// TIA Portal V18 export
FUNCTION "PLC8_910A4_8DI_8DO_IO_Update" : Void   // FC11070, LAD
{ S7_Optimized_Access := 'TRUE' }
VERSION : 0.1
// stored: AutoNumber false, IsIECCheckEnabled false, SetENOAutomatically false, UDAEnableTagReadback false
BEGIN

REGION Network 1: DIa0
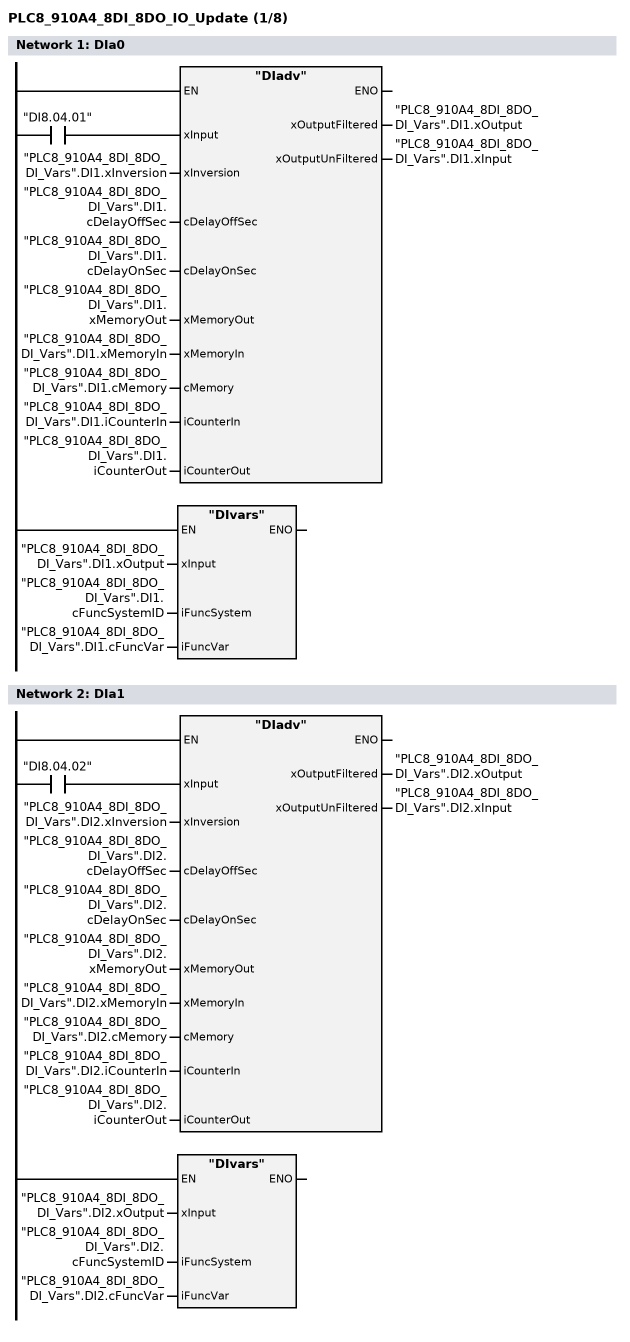
   RUNG wire#powerrail
      "DIadv"(xInput := wire#w1, xInversion := "PLC8_910A4_8DI_8DO_DI_Vars".DI1.xInversion, cDelayOffSec := "PLC8_910A4_8DI_8DO_DI_Vars".DI1.cDelayOffSec, cDelayOnSec := "PLC8_910A4_8DI_8DO_DI_Vars".DI1.cDelayOnSec, xMemoryOut := "PLC8_910A4_8DI_8DO_DI_Vars".DI1.xMemoryOut, xMemoryIn := "PLC8_910A4_8DI_8DO_DI_Vars".DI1.xMemoryIn, cMemory := "PLC8_910A4_8DI_8DO_DI_Vars".DI1.cMemory, iCounterIn := "PLC8_910A4_8DI_8DO_DI_Vars".DI1.iCounterIn, iCounterOut := "PLC8_910A4_8DI_8DO_DI_Vars".DI1.iCounterOut, xOutputFiltered => "PLC8_910A4_8DI_8DO_DI_Vars".DI1.xOutput, xOutputUnFiltered => "PLC8_910A4_8DI_8DO_DI_Vars".DI1.xInput)
   END_RUNG
   RUNG wire#powerrail
      Contact( "DI8.04.01" )
   END_RUNG wire#w1
   RUNG wire#powerrail
      "DIvars"(xInput := "PLC8_910A4_8DI_8DO_DI_Vars".DI1.xOutput, iFuncSystem := "PLC8_910A4_8DI_8DO_DI_Vars".DI1.cFuncSystemID, iFuncVar := "PLC8_910A4_8DI_8DO_DI_Vars".DI1.cFuncVar)
   END_RUNG
   // the same network as SCL:
   "DIadv"(xInput := "DI8.04.01",
           xInversion := "PLC8_910A4_8DI_8DO_DI_Vars".DI1.xInversion,
           cDelayOffSec := "PLC8_910A4_8DI_8DO_DI_Vars".DI1.cDelayOffSec,
           cDelayOnSec := "PLC8_910A4_8DI_8DO_DI_Vars".DI1.cDelayOnSec,
           xMemoryOut := "PLC8_910A4_8DI_8DO_DI_Vars".DI1.xMemoryOut,
           xMemoryIn := "PLC8_910A4_8DI_8DO_DI_Vars".DI1.xMemoryIn,
           cMemory := "PLC8_910A4_8DI_8DO_DI_Vars".DI1.cMemory,
           iCounterIn := "PLC8_910A4_8DI_8DO_DI_Vars".DI1.iCounterIn,
           iCounterOut := "PLC8_910A4_8DI_8DO_DI_Vars".DI1.iCounterOut,
           xOutputFiltered => "PLC8_910A4_8DI_8DO_DI_Vars".DI1.xOutput,
           xOutputUnFiltered => "PLC8_910A4_8DI_8DO_DI_Vars".DI1.xInput);
   "DIvars"(xInput := "PLC8_910A4_8DI_8DO_DI_Vars".DI1.xOutput,
            iFuncSystem := "PLC8_910A4_8DI_8DO_DI_Vars".DI1.cFuncSystemID,
            iFuncVar := "PLC8_910A4_8DI_8DO_DI_Vars".DI1.cFuncVar);
END_REGION

REGION Network 2: DIa1
   RUNG wire#powerrail
      "DIadv"(xInput := wire#w1, xInversion := "PLC8_910A4_8DI_8DO_DI_Vars".DI2.xInversion, cDelayOffSec := "PLC8_910A4_8DI_8DO_DI_Vars".DI2.cDelayOffSec, cDelayOnSec := "PLC8_910A4_8DI_8DO_DI_Vars".DI2.cDelayOnSec, xMemoryOut := "PLC8_910A4_8DI_8DO_DI_Vars".DI2.xMemoryOut, xMemoryIn := "PLC8_910A4_8DI_8DO_DI_Vars".DI2.xMemoryIn, cMemory := "PLC8_910A4_8DI_8DO_DI_Vars".DI2.cMemory, iCounterIn := "PLC8_910A4_8DI_8DO_DI_Vars".DI2.iCounterIn, iCounterOut := "PLC8_910A4_8DI_8DO_DI_Vars".DI2.iCounterOut, xOutputFiltered => "PLC8_910A4_8DI_8DO_DI_Vars".DI2.xOutput, xOutputUnFiltered => "PLC8_910A4_8DI_8DO_DI_Vars".DI2.xInput)
   END_RUNG
   RUNG wire#powerrail
      Contact( "DI8.04.02" )
   END_RUNG wire#w1
   RUNG wire#powerrail
      "DIvars"(xInput := "PLC8_910A4_8DI_8DO_DI_Vars".DI2.xOutput, iFuncSystem := "PLC8_910A4_8DI_8DO_DI_Vars".DI2.cFuncSystemID, iFuncVar := "PLC8_910A4_8DI_8DO_DI_Vars".DI2.cFuncVar)
   END_RUNG
   // the same network as SCL:
   "DIadv"(xInput := "DI8.04.02",
           xInversion := "PLC8_910A4_8DI_8DO_DI_Vars".DI2.xInversion,
           cDelayOffSec := "PLC8_910A4_8DI_8DO_DI_Vars".DI2.cDelayOffSec,
           cDelayOnSec := "PLC8_910A4_8DI_8DO_DI_Vars".DI2.cDelayOnSec,
           xMemoryOut := "PLC8_910A4_8DI_8DO_DI_Vars".DI2.xMemoryOut,
           xMemoryIn := "PLC8_910A4_8DI_8DO_DI_Vars".DI2.xMemoryIn,
           cMemory := "PLC8_910A4_8DI_8DO_DI_Vars".DI2.cMemory,
           iCounterIn := "PLC8_910A4_8DI_8DO_DI_Vars".DI2.iCounterIn,
           iCounterOut := "PLC8_910A4_8DI_8DO_DI_Vars".DI2.iCounterOut,
           xOutputFiltered => "PLC8_910A4_8DI_8DO_DI_Vars".DI2.xOutput,
           xOutputUnFiltered => "PLC8_910A4_8DI_8DO_DI_Vars".DI2.xInput);
   "DIvars"(xInput := "PLC8_910A4_8DI_8DO_DI_Vars".DI2.xOutput,
            iFuncSystem := "PLC8_910A4_8DI_8DO_DI_Vars".DI2.cFuncSystemID,
            iFuncVar := "PLC8_910A4_8DI_8DO_DI_Vars".DI2.cFuncVar);
END_REGION

REGION Network 3: DIa2
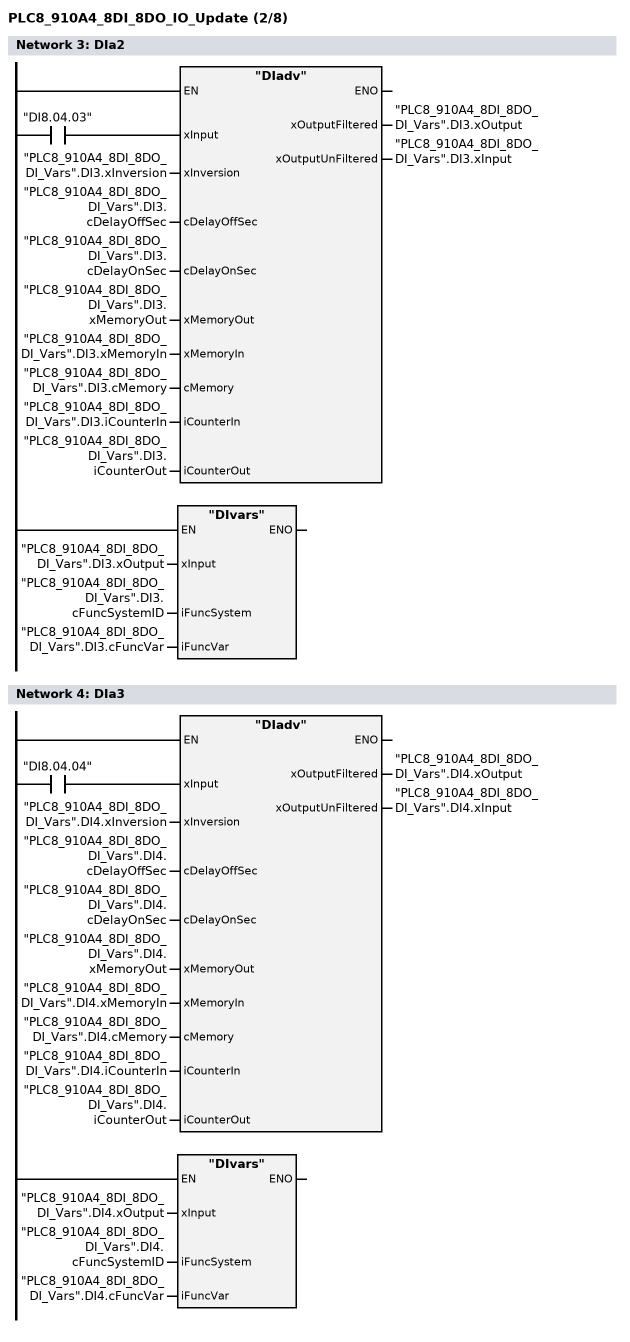
   RUNG wire#powerrail
      "DIadv"(xInput := wire#w1, xInversion := "PLC8_910A4_8DI_8DO_DI_Vars".DI3.xInversion, cDelayOffSec := "PLC8_910A4_8DI_8DO_DI_Vars".DI3.cDelayOffSec, cDelayOnSec := "PLC8_910A4_8DI_8DO_DI_Vars".DI3.cDelayOnSec, xMemoryOut := "PLC8_910A4_8DI_8DO_DI_Vars".DI3.xMemoryOut, xMemoryIn := "PLC8_910A4_8DI_8DO_DI_Vars".DI3.xMemoryIn, cMemory := "PLC8_910A4_8DI_8DO_DI_Vars".DI3.cMemory, iCounterIn := "PLC8_910A4_8DI_8DO_DI_Vars".DI3.iCounterIn, iCounterOut := "PLC8_910A4_8DI_8DO_DI_Vars".DI3.iCounterOut, xOutputFiltered => "PLC8_910A4_8DI_8DO_DI_Vars".DI3.xOutput, xOutputUnFiltered => "PLC8_910A4_8DI_8DO_DI_Vars".DI3.xInput)
   END_RUNG
   RUNG wire#powerrail
      Contact( "DI8.04.03" )
   END_RUNG wire#w1
   RUNG wire#powerrail
      "DIvars"(xInput := "PLC8_910A4_8DI_8DO_DI_Vars".DI3.xOutput, iFuncSystem := "PLC8_910A4_8DI_8DO_DI_Vars".DI3.cFuncSystemID, iFuncVar := "PLC8_910A4_8DI_8DO_DI_Vars".DI3.cFuncVar)
   END_RUNG
   // the same network as SCL:
   "DIadv"(xInput := "DI8.04.03",
           xInversion := "PLC8_910A4_8DI_8DO_DI_Vars".DI3.xInversion,
           cDelayOffSec := "PLC8_910A4_8DI_8DO_DI_Vars".DI3.cDelayOffSec,
           cDelayOnSec := "PLC8_910A4_8DI_8DO_DI_Vars".DI3.cDelayOnSec,
           xMemoryOut := "PLC8_910A4_8DI_8DO_DI_Vars".DI3.xMemoryOut,
           xMemoryIn := "PLC8_910A4_8DI_8DO_DI_Vars".DI3.xMemoryIn,
           cMemory := "PLC8_910A4_8DI_8DO_DI_Vars".DI3.cMemory,
           iCounterIn := "PLC8_910A4_8DI_8DO_DI_Vars".DI3.iCounterIn,
           iCounterOut := "PLC8_910A4_8DI_8DO_DI_Vars".DI3.iCounterOut,
           xOutputFiltered => "PLC8_910A4_8DI_8DO_DI_Vars".DI3.xOutput,
           xOutputUnFiltered => "PLC8_910A4_8DI_8DO_DI_Vars".DI3.xInput);
   "DIvars"(xInput := "PLC8_910A4_8DI_8DO_DI_Vars".DI3.xOutput,
            iFuncSystem := "PLC8_910A4_8DI_8DO_DI_Vars".DI3.cFuncSystemID,
            iFuncVar := "PLC8_910A4_8DI_8DO_DI_Vars".DI3.cFuncVar);
END_REGION

REGION Network 4: DIa3
   RUNG wire#powerrail
      "DIadv"(xInput := wire#w1, xInversion := "PLC8_910A4_8DI_8DO_DI_Vars".DI4.xInversion, cDelayOffSec := "PLC8_910A4_8DI_8DO_DI_Vars".DI4.cDelayOffSec, cDelayOnSec := "PLC8_910A4_8DI_8DO_DI_Vars".DI4.cDelayOnSec, xMemoryOut := "PLC8_910A4_8DI_8DO_DI_Vars".DI4.xMemoryOut, xMemoryIn := "PLC8_910A4_8DI_8DO_DI_Vars".DI4.xMemoryIn, cMemory := "PLC8_910A4_8DI_8DO_DI_Vars".DI4.cMemory, iCounterIn := "PLC8_910A4_8DI_8DO_DI_Vars".DI4.iCounterIn, iCounterOut := "PLC8_910A4_8DI_8DO_DI_Vars".DI4.iCounterOut, xOutputFiltered => "PLC8_910A4_8DI_8DO_DI_Vars".DI4.xOutput, xOutputUnFiltered => "PLC8_910A4_8DI_8DO_DI_Vars".DI4.xInput)
   END_RUNG
   RUNG wire#powerrail
      Contact( "DI8.04.04" )
   END_RUNG wire#w1
   RUNG wire#powerrail
      "DIvars"(xInput := "PLC8_910A4_8DI_8DO_DI_Vars".DI4.xOutput, iFuncSystem := "PLC8_910A4_8DI_8DO_DI_Vars".DI4.cFuncSystemID, iFuncVar := "PLC8_910A4_8DI_8DO_DI_Vars".DI4.cFuncVar)
   END_RUNG
   // the same network as SCL:
   "DIadv"(xInput := "DI8.04.04",
           xInversion := "PLC8_910A4_8DI_8DO_DI_Vars".DI4.xInversion,
           cDelayOffSec := "PLC8_910A4_8DI_8DO_DI_Vars".DI4.cDelayOffSec,
           cDelayOnSec := "PLC8_910A4_8DI_8DO_DI_Vars".DI4.cDelayOnSec,
           xMemoryOut := "PLC8_910A4_8DI_8DO_DI_Vars".DI4.xMemoryOut,
           xMemoryIn := "PLC8_910A4_8DI_8DO_DI_Vars".DI4.xMemoryIn,
           cMemory := "PLC8_910A4_8DI_8DO_DI_Vars".DI4.cMemory,
           iCounterIn := "PLC8_910A4_8DI_8DO_DI_Vars".DI4.iCounterIn,
           iCounterOut := "PLC8_910A4_8DI_8DO_DI_Vars".DI4.iCounterOut,
           xOutputFiltered => "PLC8_910A4_8DI_8DO_DI_Vars".DI4.xOutput,
           xOutputUnFiltered => "PLC8_910A4_8DI_8DO_DI_Vars".DI4.xInput);
   "DIvars"(xInput := "PLC8_910A4_8DI_8DO_DI_Vars".DI4.xOutput,
            iFuncSystem := "PLC8_910A4_8DI_8DO_DI_Vars".DI4.cFuncSystemID,
            iFuncVar := "PLC8_910A4_8DI_8DO_DI_Vars".DI4.cFuncVar);
END_REGION

REGION Network 5: DIa4
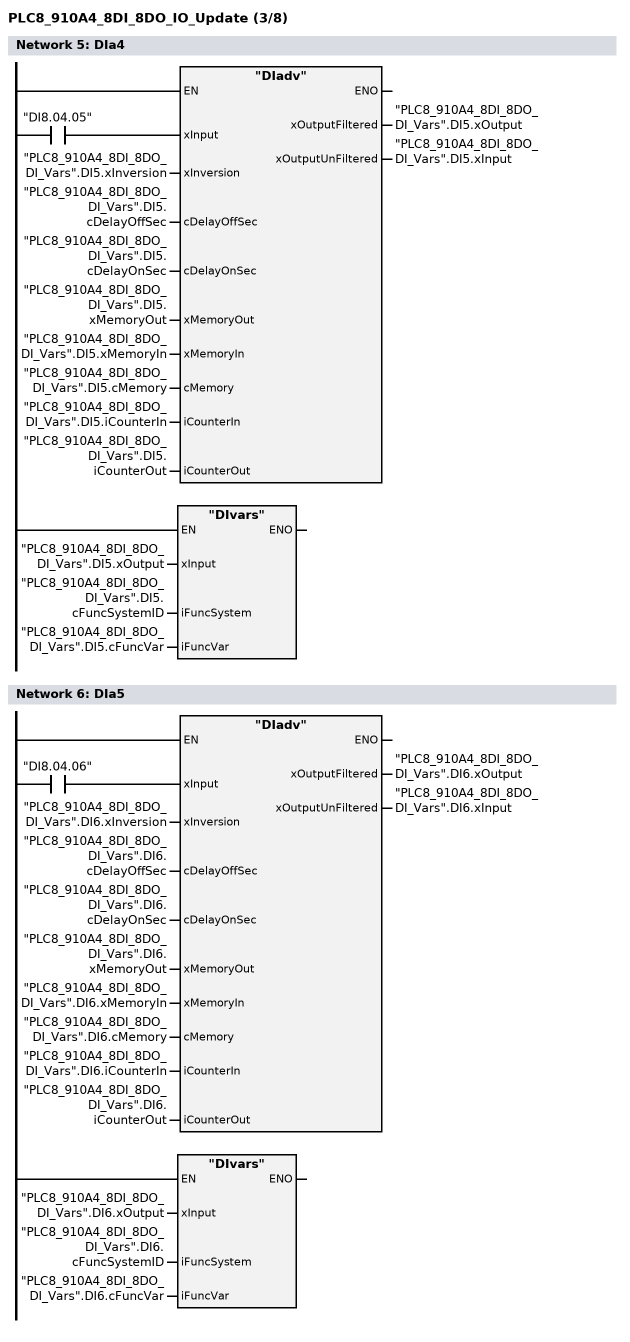
   RUNG wire#powerrail
      "DIadv"(xInput := wire#w1, xInversion := "PLC8_910A4_8DI_8DO_DI_Vars".DI5.xInversion, cDelayOffSec := "PLC8_910A4_8DI_8DO_DI_Vars".DI5.cDelayOffSec, cDelayOnSec := "PLC8_910A4_8DI_8DO_DI_Vars".DI5.cDelayOnSec, xMemoryOut := "PLC8_910A4_8DI_8DO_DI_Vars".DI5.xMemoryOut, xMemoryIn := "PLC8_910A4_8DI_8DO_DI_Vars".DI5.xMemoryIn, cMemory := "PLC8_910A4_8DI_8DO_DI_Vars".DI5.cMemory, iCounterIn := "PLC8_910A4_8DI_8DO_DI_Vars".DI5.iCounterIn, iCounterOut := "PLC8_910A4_8DI_8DO_DI_Vars".DI5.iCounterOut, xOutputFiltered => "PLC8_910A4_8DI_8DO_DI_Vars".DI5.xOutput, xOutputUnFiltered => "PLC8_910A4_8DI_8DO_DI_Vars".DI5.xInput)
   END_RUNG
   RUNG wire#powerrail
      Contact( "DI8.04.05" )
   END_RUNG wire#w1
   RUNG wire#powerrail
      "DIvars"(xInput := "PLC8_910A4_8DI_8DO_DI_Vars".DI5.xOutput, iFuncSystem := "PLC8_910A4_8DI_8DO_DI_Vars".DI5.cFuncSystemID, iFuncVar := "PLC8_910A4_8DI_8DO_DI_Vars".DI5.cFuncVar)
   END_RUNG
   // the same network as SCL:
   "DIadv"(xInput := "DI8.04.05",
           xInversion := "PLC8_910A4_8DI_8DO_DI_Vars".DI5.xInversion,
           cDelayOffSec := "PLC8_910A4_8DI_8DO_DI_Vars".DI5.cDelayOffSec,
           cDelayOnSec := "PLC8_910A4_8DI_8DO_DI_Vars".DI5.cDelayOnSec,
           xMemoryOut := "PLC8_910A4_8DI_8DO_DI_Vars".DI5.xMemoryOut,
           xMemoryIn := "PLC8_910A4_8DI_8DO_DI_Vars".DI5.xMemoryIn,
           cMemory := "PLC8_910A4_8DI_8DO_DI_Vars".DI5.cMemory,
           iCounterIn := "PLC8_910A4_8DI_8DO_DI_Vars".DI5.iCounterIn,
           iCounterOut := "PLC8_910A4_8DI_8DO_DI_Vars".DI5.iCounterOut,
           xOutputFiltered => "PLC8_910A4_8DI_8DO_DI_Vars".DI5.xOutput,
           xOutputUnFiltered => "PLC8_910A4_8DI_8DO_DI_Vars".DI5.xInput);
   "DIvars"(xInput := "PLC8_910A4_8DI_8DO_DI_Vars".DI5.xOutput,
            iFuncSystem := "PLC8_910A4_8DI_8DO_DI_Vars".DI5.cFuncSystemID,
            iFuncVar := "PLC8_910A4_8DI_8DO_DI_Vars".DI5.cFuncVar);
END_REGION

REGION Network 6: DIa5
   RUNG wire#powerrail
      "DIadv"(xInput := wire#w1, xInversion := "PLC8_910A4_8DI_8DO_DI_Vars".DI6.xInversion, cDelayOffSec := "PLC8_910A4_8DI_8DO_DI_Vars".DI6.cDelayOffSec, cDelayOnSec := "PLC8_910A4_8DI_8DO_DI_Vars".DI6.cDelayOnSec, xMemoryOut := "PLC8_910A4_8DI_8DO_DI_Vars".DI6.xMemoryOut, xMemoryIn := "PLC8_910A4_8DI_8DO_DI_Vars".DI6.xMemoryIn, cMemory := "PLC8_910A4_8DI_8DO_DI_Vars".DI6.cMemory, iCounterIn := "PLC8_910A4_8DI_8DO_DI_Vars".DI6.iCounterIn, iCounterOut := "PLC8_910A4_8DI_8DO_DI_Vars".DI6.iCounterOut, xOutputFiltered => "PLC8_910A4_8DI_8DO_DI_Vars".DI6.xOutput, xOutputUnFiltered => "PLC8_910A4_8DI_8DO_DI_Vars".DI6.xInput)
   END_RUNG
   RUNG wire#powerrail
      Contact( "DI8.04.06" )
   END_RUNG wire#w1
   RUNG wire#powerrail
      "DIvars"(xInput := "PLC8_910A4_8DI_8DO_DI_Vars".DI6.xOutput, iFuncSystem := "PLC8_910A4_8DI_8DO_DI_Vars".DI6.cFuncSystemID, iFuncVar := "PLC8_910A4_8DI_8DO_DI_Vars".DI6.cFuncVar)
   END_RUNG
   // the same network as SCL:
   "DIadv"(xInput := "DI8.04.06",
           xInversion := "PLC8_910A4_8DI_8DO_DI_Vars".DI6.xInversion,
           cDelayOffSec := "PLC8_910A4_8DI_8DO_DI_Vars".DI6.cDelayOffSec,
           cDelayOnSec := "PLC8_910A4_8DI_8DO_DI_Vars".DI6.cDelayOnSec,
           xMemoryOut := "PLC8_910A4_8DI_8DO_DI_Vars".DI6.xMemoryOut,
           xMemoryIn := "PLC8_910A4_8DI_8DO_DI_Vars".DI6.xMemoryIn,
           cMemory := "PLC8_910A4_8DI_8DO_DI_Vars".DI6.cMemory,
           iCounterIn := "PLC8_910A4_8DI_8DO_DI_Vars".DI6.iCounterIn,
           iCounterOut := "PLC8_910A4_8DI_8DO_DI_Vars".DI6.iCounterOut,
           xOutputFiltered => "PLC8_910A4_8DI_8DO_DI_Vars".DI6.xOutput,
           xOutputUnFiltered => "PLC8_910A4_8DI_8DO_DI_Vars".DI6.xInput);
   "DIvars"(xInput := "PLC8_910A4_8DI_8DO_DI_Vars".DI6.xOutput,
            iFuncSystem := "PLC8_910A4_8DI_8DO_DI_Vars".DI6.cFuncSystemID,
            iFuncVar := "PLC8_910A4_8DI_8DO_DI_Vars".DI6.cFuncVar);
END_REGION

REGION Network 7: DIa6
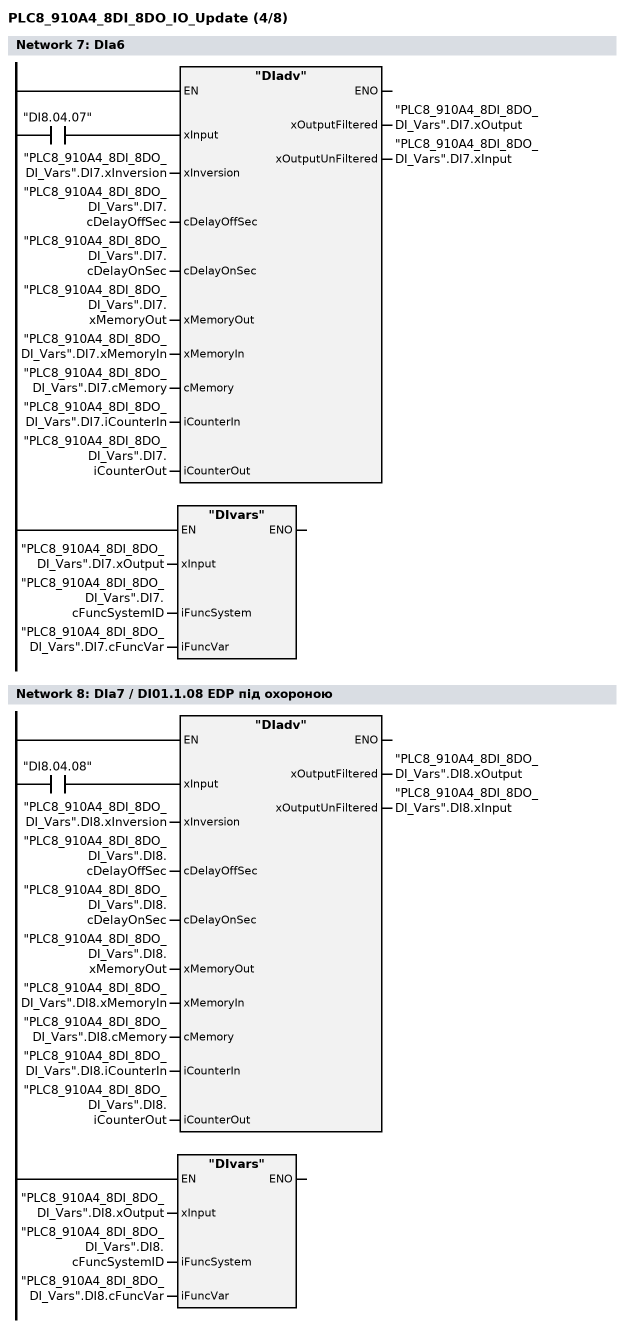
   RUNG wire#powerrail
      "DIadv"(xInput := wire#w1, xInversion := "PLC8_910A4_8DI_8DO_DI_Vars".DI7.xInversion, cDelayOffSec := "PLC8_910A4_8DI_8DO_DI_Vars".DI7.cDelayOffSec, cDelayOnSec := "PLC8_910A4_8DI_8DO_DI_Vars".DI7.cDelayOnSec, xMemoryOut := "PLC8_910A4_8DI_8DO_DI_Vars".DI7.xMemoryOut, xMemoryIn := "PLC8_910A4_8DI_8DO_DI_Vars".DI7.xMemoryIn, cMemory := "PLC8_910A4_8DI_8DO_DI_Vars".DI7.cMemory, iCounterIn := "PLC8_910A4_8DI_8DO_DI_Vars".DI7.iCounterIn, iCounterOut := "PLC8_910A4_8DI_8DO_DI_Vars".DI7.iCounterOut, xOutputFiltered => "PLC8_910A4_8DI_8DO_DI_Vars".DI7.xOutput, xOutputUnFiltered => "PLC8_910A4_8DI_8DO_DI_Vars".DI7.xInput)
   END_RUNG
   RUNG wire#powerrail
      Contact( "DI8.04.07" )
   END_RUNG wire#w1
   RUNG wire#powerrail
      "DIvars"(xInput := "PLC8_910A4_8DI_8DO_DI_Vars".DI7.xOutput, iFuncSystem := "PLC8_910A4_8DI_8DO_DI_Vars".DI7.cFuncSystemID, iFuncVar := "PLC8_910A4_8DI_8DO_DI_Vars".DI7.cFuncVar)
   END_RUNG
   // the same network as SCL:
   "DIadv"(xInput := "DI8.04.07",
           xInversion := "PLC8_910A4_8DI_8DO_DI_Vars".DI7.xInversion,
           cDelayOffSec := "PLC8_910A4_8DI_8DO_DI_Vars".DI7.cDelayOffSec,
           cDelayOnSec := "PLC8_910A4_8DI_8DO_DI_Vars".DI7.cDelayOnSec,
           xMemoryOut := "PLC8_910A4_8DI_8DO_DI_Vars".DI7.xMemoryOut,
           xMemoryIn := "PLC8_910A4_8DI_8DO_DI_Vars".DI7.xMemoryIn,
           cMemory := "PLC8_910A4_8DI_8DO_DI_Vars".DI7.cMemory,
           iCounterIn := "PLC8_910A4_8DI_8DO_DI_Vars".DI7.iCounterIn,
           iCounterOut := "PLC8_910A4_8DI_8DO_DI_Vars".DI7.iCounterOut,
           xOutputFiltered => "PLC8_910A4_8DI_8DO_DI_Vars".DI7.xOutput,
           xOutputUnFiltered => "PLC8_910A4_8DI_8DO_DI_Vars".DI7.xInput);
   "DIvars"(xInput := "PLC8_910A4_8DI_8DO_DI_Vars".DI7.xOutput,
            iFuncSystem := "PLC8_910A4_8DI_8DO_DI_Vars".DI7.cFuncSystemID,
            iFuncVar := "PLC8_910A4_8DI_8DO_DI_Vars".DI7.cFuncVar);
END_REGION

REGION Network 8: DIa7 / DI01.1.08 EDP під охороною
   RUNG wire#powerrail
      "DIadv"(xInput := wire#w1, xInversion := "PLC8_910A4_8DI_8DO_DI_Vars".DI8.xInversion, cDelayOffSec := "PLC8_910A4_8DI_8DO_DI_Vars".DI8.cDelayOffSec, cDelayOnSec := "PLC8_910A4_8DI_8DO_DI_Vars".DI8.cDelayOnSec, xMemoryOut := "PLC8_910A4_8DI_8DO_DI_Vars".DI8.xMemoryOut, xMemoryIn := "PLC8_910A4_8DI_8DO_DI_Vars".DI8.xMemoryIn, cMemory := "PLC8_910A4_8DI_8DO_DI_Vars".DI8.cMemory, iCounterIn := "PLC8_910A4_8DI_8DO_DI_Vars".DI8.iCounterIn, iCounterOut := "PLC8_910A4_8DI_8DO_DI_Vars".DI8.iCounterOut, xOutputFiltered => "PLC8_910A4_8DI_8DO_DI_Vars".DI8.xOutput, xOutputUnFiltered => "PLC8_910A4_8DI_8DO_DI_Vars".DI8.xInput)
   END_RUNG
   RUNG wire#powerrail
      Contact( "DI8.04.08" )
   END_RUNG wire#w1
   RUNG wire#powerrail
      "DIvars"(xInput := "PLC8_910A4_8DI_8DO_DI_Vars".DI8.xOutput, iFuncSystem := "PLC8_910A4_8DI_8DO_DI_Vars".DI8.cFuncSystemID, iFuncVar := "PLC8_910A4_8DI_8DO_DI_Vars".DI8.cFuncVar)
   END_RUNG
   // the same network as SCL:
   "DIadv"(xInput := "DI8.04.08",
           xInversion := "PLC8_910A4_8DI_8DO_DI_Vars".DI8.xInversion,
           cDelayOffSec := "PLC8_910A4_8DI_8DO_DI_Vars".DI8.cDelayOffSec,
           cDelayOnSec := "PLC8_910A4_8DI_8DO_DI_Vars".DI8.cDelayOnSec,
           xMemoryOut := "PLC8_910A4_8DI_8DO_DI_Vars".DI8.xMemoryOut,
           xMemoryIn := "PLC8_910A4_8DI_8DO_DI_Vars".DI8.xMemoryIn,
           cMemory := "PLC8_910A4_8DI_8DO_DI_Vars".DI8.cMemory,
           iCounterIn := "PLC8_910A4_8DI_8DO_DI_Vars".DI8.iCounterIn,
           iCounterOut := "PLC8_910A4_8DI_8DO_DI_Vars".DI8.iCounterOut,
           xOutputFiltered => "PLC8_910A4_8DI_8DO_DI_Vars".DI8.xOutput,
           xOutputUnFiltered => "PLC8_910A4_8DI_8DO_DI_Vars".DI8.xInput);
   "DIvars"(xInput := "PLC8_910A4_8DI_8DO_DI_Vars".DI8.xOutput,
            iFuncSystem := "PLC8_910A4_8DI_8DO_DI_Vars".DI8.cFuncSystemID,
            iFuncVar := "PLC8_910A4_8DI_8DO_DI_Vars".DI8.cFuncVar);
END_REGION

REGION Network 9: DQa0
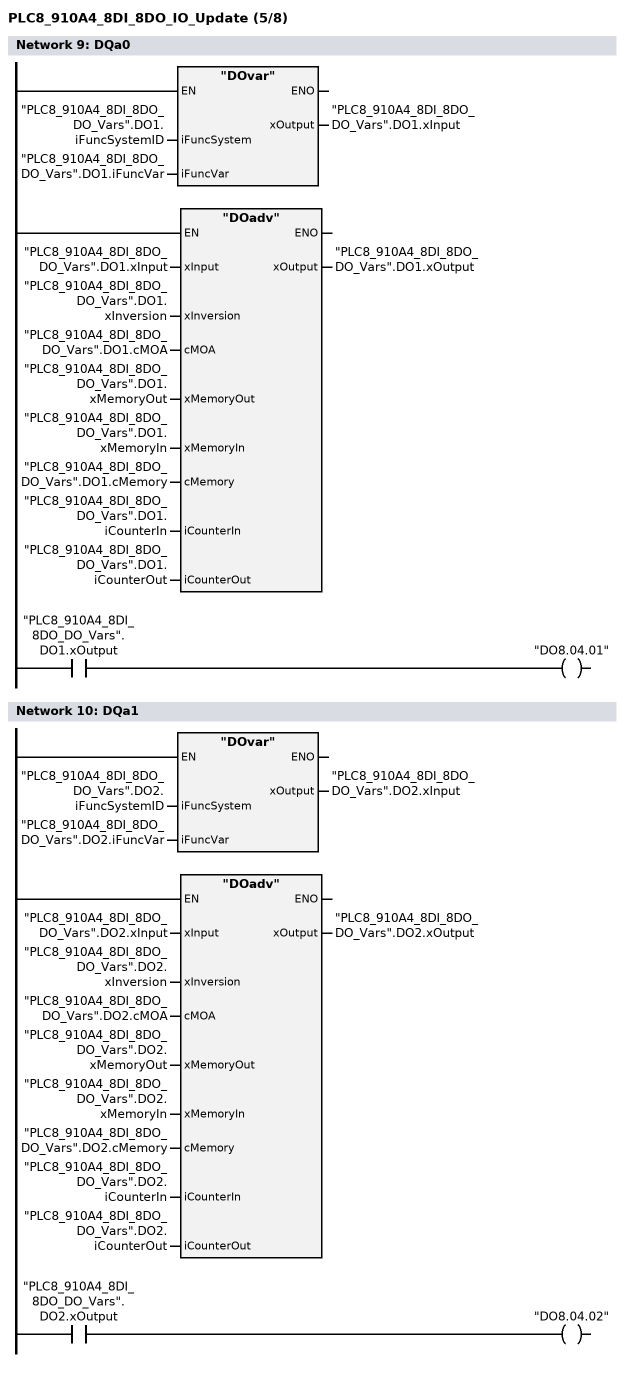
   RUNG wire#powerrail
      "DOvar"(iFuncSystem := "PLC8_910A4_8DI_8DO_DO_Vars".DO1.iFuncSystemID, iFuncVar := "PLC8_910A4_8DI_8DO_DO_Vars".DO1.iFuncVar, xOutput => "PLC8_910A4_8DI_8DO_DO_Vars".DO1.xInput)
   END_RUNG
   RUNG wire#powerrail
      "DOadv"(xInput := "PLC8_910A4_8DI_8DO_DO_Vars".DO1.xInput, xInversion := "PLC8_910A4_8DI_8DO_DO_Vars".DO1.xInversion, cMOA := "PLC8_910A4_8DI_8DO_DO_Vars".DO1.cMOA, xMemoryOut := "PLC8_910A4_8DI_8DO_DO_Vars".DO1.xMemoryOut, xMemoryIn := "PLC8_910A4_8DI_8DO_DO_Vars".DO1.xMemoryIn, cMemory := "PLC8_910A4_8DI_8DO_DO_Vars".DO1.cMemory, iCounterIn := "PLC8_910A4_8DI_8DO_DO_Vars".DO1.iCounterIn, iCounterOut := "PLC8_910A4_8DI_8DO_DO_Vars".DO1.iCounterOut, xOutput => "PLC8_910A4_8DI_8DO_DO_Vars".DO1.xOutput)
   END_RUNG
   RUNG wire#powerrail
      Contact( "PLC8_910A4_8DI_8DO_DO_Vars".DO1.xOutput )
      Coil( "DO8.04.01" )
   END_RUNG
   // the same network as SCL:
   "DOvar"(iFuncSystem := "PLC8_910A4_8DI_8DO_DO_Vars".DO1.iFuncSystemID,
           iFuncVar := "PLC8_910A4_8DI_8DO_DO_Vars".DO1.iFuncVar,
           xOutput => "PLC8_910A4_8DI_8DO_DO_Vars".DO1.xInput);
   "DOadv"(xInput := "PLC8_910A4_8DI_8DO_DO_Vars".DO1.xInput,
           xInversion := "PLC8_910A4_8DI_8DO_DO_Vars".DO1.xInversion,
           cMOA := "PLC8_910A4_8DI_8DO_DO_Vars".DO1.cMOA,
           xMemoryOut := "PLC8_910A4_8DI_8DO_DO_Vars".DO1.xMemoryOut,
           xMemoryIn := "PLC8_910A4_8DI_8DO_DO_Vars".DO1.xMemoryIn,
           cMemory := "PLC8_910A4_8DI_8DO_DO_Vars".DO1.cMemory,
           iCounterIn := "PLC8_910A4_8DI_8DO_DO_Vars".DO1.iCounterIn,
           iCounterOut := "PLC8_910A4_8DI_8DO_DO_Vars".DO1.iCounterOut,
           xOutput => "PLC8_910A4_8DI_8DO_DO_Vars".DO1.xOutput);
   "DO8.04.01" := "PLC8_910A4_8DI_8DO_DO_Vars".DO1.xOutput;
END_REGION

REGION Network 10: DQa1
   RUNG wire#powerrail
      "DOvar"(iFuncSystem := "PLC8_910A4_8DI_8DO_DO_Vars".DO2.iFuncSystemID, iFuncVar := "PLC8_910A4_8DI_8DO_DO_Vars".DO2.iFuncVar, xOutput => "PLC8_910A4_8DI_8DO_DO_Vars".DO2.xInput)
   END_RUNG
   RUNG wire#powerrail
      "DOadv"(xInput := "PLC8_910A4_8DI_8DO_DO_Vars".DO2.xInput, xInversion := "PLC8_910A4_8DI_8DO_DO_Vars".DO2.xInversion, cMOA := "PLC8_910A4_8DI_8DO_DO_Vars".DO2.cMOA, xMemoryOut := "PLC8_910A4_8DI_8DO_DO_Vars".DO2.xMemoryOut, xMemoryIn := "PLC8_910A4_8DI_8DO_DO_Vars".DO2.xMemoryIn, cMemory := "PLC8_910A4_8DI_8DO_DO_Vars".DO2.cMemory, iCounterIn := "PLC8_910A4_8DI_8DO_DO_Vars".DO2.iCounterIn, iCounterOut := "PLC8_910A4_8DI_8DO_DO_Vars".DO2.iCounterOut, xOutput => "PLC8_910A4_8DI_8DO_DO_Vars".DO2.xOutput)
   END_RUNG
   RUNG wire#powerrail
      Contact( "PLC8_910A4_8DI_8DO_DO_Vars".DO2.xOutput )
      Coil( "DO8.04.02" )
   END_RUNG
   // the same network as SCL:
   "DOvar"(iFuncSystem := "PLC8_910A4_8DI_8DO_DO_Vars".DO2.iFuncSystemID,
           iFuncVar := "PLC8_910A4_8DI_8DO_DO_Vars".DO2.iFuncVar,
           xOutput => "PLC8_910A4_8DI_8DO_DO_Vars".DO2.xInput);
   "DOadv"(xInput := "PLC8_910A4_8DI_8DO_DO_Vars".DO2.xInput,
           xInversion := "PLC8_910A4_8DI_8DO_DO_Vars".DO2.xInversion,
           cMOA := "PLC8_910A4_8DI_8DO_DO_Vars".DO2.cMOA,
           xMemoryOut := "PLC8_910A4_8DI_8DO_DO_Vars".DO2.xMemoryOut,
           xMemoryIn := "PLC8_910A4_8DI_8DO_DO_Vars".DO2.xMemoryIn,
           cMemory := "PLC8_910A4_8DI_8DO_DO_Vars".DO2.cMemory,
           iCounterIn := "PLC8_910A4_8DI_8DO_DO_Vars".DO2.iCounterIn,
           iCounterOut := "PLC8_910A4_8DI_8DO_DO_Vars".DO2.iCounterOut,
           xOutput => "PLC8_910A4_8DI_8DO_DO_Vars".DO2.xOutput);
   "DO8.04.02" := "PLC8_910A4_8DI_8DO_DO_Vars".DO2.xOutput;
END_REGION

REGION Network 11: DQa2
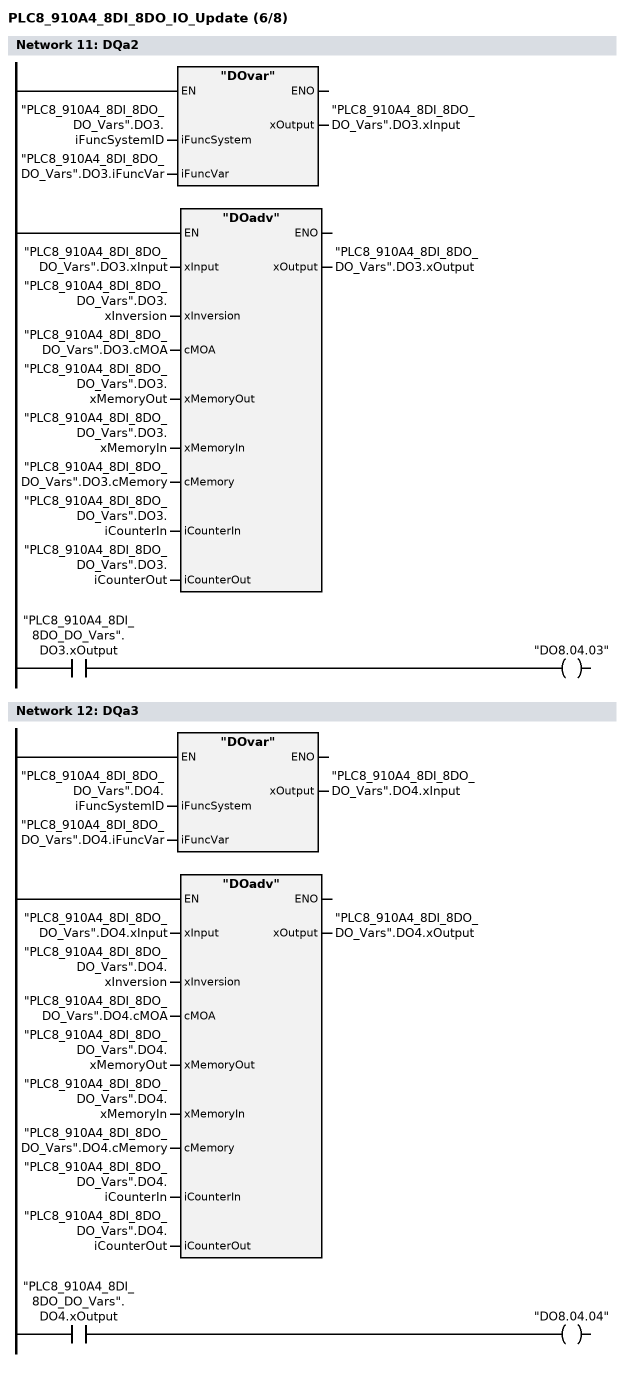
   RUNG wire#powerrail
      "DOvar"(iFuncSystem := "PLC8_910A4_8DI_8DO_DO_Vars".DO3.iFuncSystemID, iFuncVar := "PLC8_910A4_8DI_8DO_DO_Vars".DO3.iFuncVar, xOutput => "PLC8_910A4_8DI_8DO_DO_Vars".DO3.xInput)
   END_RUNG
   RUNG wire#powerrail
      "DOadv"(xInput := "PLC8_910A4_8DI_8DO_DO_Vars".DO3.xInput, xInversion := "PLC8_910A4_8DI_8DO_DO_Vars".DO3.xInversion, cMOA := "PLC8_910A4_8DI_8DO_DO_Vars".DO3.cMOA, xMemoryOut := "PLC8_910A4_8DI_8DO_DO_Vars".DO3.xMemoryOut, xMemoryIn := "PLC8_910A4_8DI_8DO_DO_Vars".DO3.xMemoryIn, cMemory := "PLC8_910A4_8DI_8DO_DO_Vars".DO3.cMemory, iCounterIn := "PLC8_910A4_8DI_8DO_DO_Vars".DO3.iCounterIn, iCounterOut := "PLC8_910A4_8DI_8DO_DO_Vars".DO3.iCounterOut, xOutput => "PLC8_910A4_8DI_8DO_DO_Vars".DO3.xOutput)
   END_RUNG
   RUNG wire#powerrail
      Contact( "PLC8_910A4_8DI_8DO_DO_Vars".DO3.xOutput )
      Coil( "DO8.04.03" )
   END_RUNG
   // the same network as SCL:
   "DOvar"(iFuncSystem := "PLC8_910A4_8DI_8DO_DO_Vars".DO3.iFuncSystemID,
           iFuncVar := "PLC8_910A4_8DI_8DO_DO_Vars".DO3.iFuncVar,
           xOutput => "PLC8_910A4_8DI_8DO_DO_Vars".DO3.xInput);
   "DOadv"(xInput := "PLC8_910A4_8DI_8DO_DO_Vars".DO3.xInput,
           xInversion := "PLC8_910A4_8DI_8DO_DO_Vars".DO3.xInversion,
           cMOA := "PLC8_910A4_8DI_8DO_DO_Vars".DO3.cMOA,
           xMemoryOut := "PLC8_910A4_8DI_8DO_DO_Vars".DO3.xMemoryOut,
           xMemoryIn := "PLC8_910A4_8DI_8DO_DO_Vars".DO3.xMemoryIn,
           cMemory := "PLC8_910A4_8DI_8DO_DO_Vars".DO3.cMemory,
           iCounterIn := "PLC8_910A4_8DI_8DO_DO_Vars".DO3.iCounterIn,
           iCounterOut := "PLC8_910A4_8DI_8DO_DO_Vars".DO3.iCounterOut,
           xOutput => "PLC8_910A4_8DI_8DO_DO_Vars".DO3.xOutput);
   "DO8.04.03" := "PLC8_910A4_8DI_8DO_DO_Vars".DO3.xOutput;
END_REGION

REGION Network 12: DQa3
   RUNG wire#powerrail
      "DOvar"(iFuncSystem := "PLC8_910A4_8DI_8DO_DO_Vars".DO4.iFuncSystemID, iFuncVar := "PLC8_910A4_8DI_8DO_DO_Vars".DO4.iFuncVar, xOutput => "PLC8_910A4_8DI_8DO_DO_Vars".DO4.xInput)
   END_RUNG
   RUNG wire#powerrail
      "DOadv"(xInput := "PLC8_910A4_8DI_8DO_DO_Vars".DO4.xInput, xInversion := "PLC8_910A4_8DI_8DO_DO_Vars".DO4.xInversion, cMOA := "PLC8_910A4_8DI_8DO_DO_Vars".DO4.cMOA, xMemoryOut := "PLC8_910A4_8DI_8DO_DO_Vars".DO4.xMemoryOut, xMemoryIn := "PLC8_910A4_8DI_8DO_DO_Vars".DO4.xMemoryIn, cMemory := "PLC8_910A4_8DI_8DO_DO_Vars".DO4.cMemory, iCounterIn := "PLC8_910A4_8DI_8DO_DO_Vars".DO4.iCounterIn, iCounterOut := "PLC8_910A4_8DI_8DO_DO_Vars".DO4.iCounterOut, xOutput => "PLC8_910A4_8DI_8DO_DO_Vars".DO4.xOutput)
   END_RUNG
   RUNG wire#powerrail
      Contact( "PLC8_910A4_8DI_8DO_DO_Vars".DO4.xOutput )
      Coil( "DO8.04.04" )
   END_RUNG
   // the same network as SCL:
   "DOvar"(iFuncSystem := "PLC8_910A4_8DI_8DO_DO_Vars".DO4.iFuncSystemID,
           iFuncVar := "PLC8_910A4_8DI_8DO_DO_Vars".DO4.iFuncVar,
           xOutput => "PLC8_910A4_8DI_8DO_DO_Vars".DO4.xInput);
   "DOadv"(xInput := "PLC8_910A4_8DI_8DO_DO_Vars".DO4.xInput,
           xInversion := "PLC8_910A4_8DI_8DO_DO_Vars".DO4.xInversion,
           cMOA := "PLC8_910A4_8DI_8DO_DO_Vars".DO4.cMOA,
           xMemoryOut := "PLC8_910A4_8DI_8DO_DO_Vars".DO4.xMemoryOut,
           xMemoryIn := "PLC8_910A4_8DI_8DO_DO_Vars".DO4.xMemoryIn,
           cMemory := "PLC8_910A4_8DI_8DO_DO_Vars".DO4.cMemory,
           iCounterIn := "PLC8_910A4_8DI_8DO_DO_Vars".DO4.iCounterIn,
           iCounterOut := "PLC8_910A4_8DI_8DO_DO_Vars".DO4.iCounterOut,
           xOutput => "PLC8_910A4_8DI_8DO_DO_Vars".DO4.xOutput);
   "DO8.04.04" := "PLC8_910A4_8DI_8DO_DO_Vars".DO4.xOutput;
END_REGION

REGION Network 13: DQa4
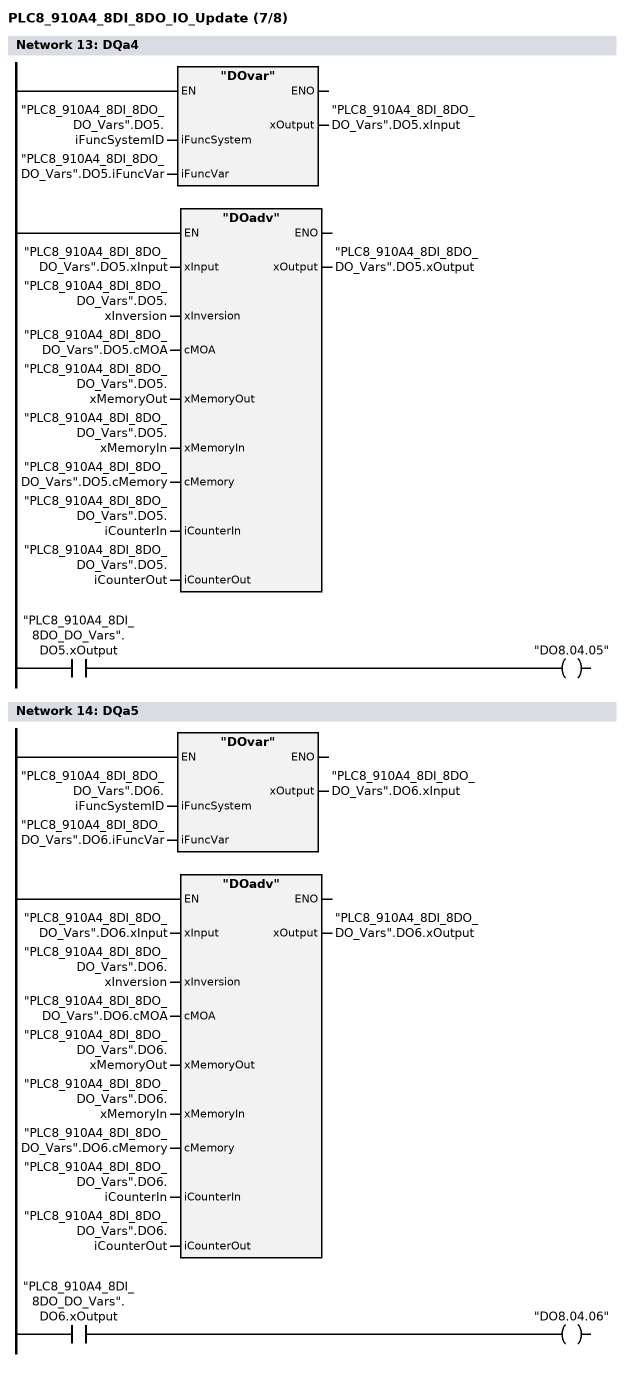
   RUNG wire#powerrail
      "DOvar"(iFuncSystem := "PLC8_910A4_8DI_8DO_DO_Vars".DO5.iFuncSystemID, iFuncVar := "PLC8_910A4_8DI_8DO_DO_Vars".DO5.iFuncVar, xOutput => "PLC8_910A4_8DI_8DO_DO_Vars".DO5.xInput)
   END_RUNG
   RUNG wire#powerrail
      "DOadv"(xInput := "PLC8_910A4_8DI_8DO_DO_Vars".DO5.xInput, xInversion := "PLC8_910A4_8DI_8DO_DO_Vars".DO5.xInversion, cMOA := "PLC8_910A4_8DI_8DO_DO_Vars".DO5.cMOA, xMemoryOut := "PLC8_910A4_8DI_8DO_DO_Vars".DO5.xMemoryOut, xMemoryIn := "PLC8_910A4_8DI_8DO_DO_Vars".DO5.xMemoryIn, cMemory := "PLC8_910A4_8DI_8DO_DO_Vars".DO5.cMemory, iCounterIn := "PLC8_910A4_8DI_8DO_DO_Vars".DO5.iCounterIn, iCounterOut := "PLC8_910A4_8DI_8DO_DO_Vars".DO5.iCounterOut, xOutput => "PLC8_910A4_8DI_8DO_DO_Vars".DO5.xOutput)
   END_RUNG
   RUNG wire#powerrail
      Contact( "PLC8_910A4_8DI_8DO_DO_Vars".DO5.xOutput )
      Coil( "DO8.04.05" )
   END_RUNG
   // the same network as SCL:
   "DOvar"(iFuncSystem := "PLC8_910A4_8DI_8DO_DO_Vars".DO5.iFuncSystemID,
           iFuncVar := "PLC8_910A4_8DI_8DO_DO_Vars".DO5.iFuncVar,
           xOutput => "PLC8_910A4_8DI_8DO_DO_Vars".DO5.xInput);
   "DOadv"(xInput := "PLC8_910A4_8DI_8DO_DO_Vars".DO5.xInput,
           xInversion := "PLC8_910A4_8DI_8DO_DO_Vars".DO5.xInversion,
           cMOA := "PLC8_910A4_8DI_8DO_DO_Vars".DO5.cMOA,
           xMemoryOut := "PLC8_910A4_8DI_8DO_DO_Vars".DO5.xMemoryOut,
           xMemoryIn := "PLC8_910A4_8DI_8DO_DO_Vars".DO5.xMemoryIn,
           cMemory := "PLC8_910A4_8DI_8DO_DO_Vars".DO5.cMemory,
           iCounterIn := "PLC8_910A4_8DI_8DO_DO_Vars".DO5.iCounterIn,
           iCounterOut := "PLC8_910A4_8DI_8DO_DO_Vars".DO5.iCounterOut,
           xOutput => "PLC8_910A4_8DI_8DO_DO_Vars".DO5.xOutput);
   "DO8.04.05" := "PLC8_910A4_8DI_8DO_DO_Vars".DO5.xOutput;
END_REGION

REGION Network 14: DQa5
   RUNG wire#powerrail
      "DOvar"(iFuncSystem := "PLC8_910A4_8DI_8DO_DO_Vars".DO6.iFuncSystemID, iFuncVar := "PLC8_910A4_8DI_8DO_DO_Vars".DO6.iFuncVar, xOutput => "PLC8_910A4_8DI_8DO_DO_Vars".DO6.xInput)
   END_RUNG
   RUNG wire#powerrail
      "DOadv"(xInput := "PLC8_910A4_8DI_8DO_DO_Vars".DO6.xInput, xInversion := "PLC8_910A4_8DI_8DO_DO_Vars".DO6.xInversion, cMOA := "PLC8_910A4_8DI_8DO_DO_Vars".DO6.cMOA, xMemoryOut := "PLC8_910A4_8DI_8DO_DO_Vars".DO6.xMemoryOut, xMemoryIn := "PLC8_910A4_8DI_8DO_DO_Vars".DO6.xMemoryIn, cMemory := "PLC8_910A4_8DI_8DO_DO_Vars".DO6.cMemory, iCounterIn := "PLC8_910A4_8DI_8DO_DO_Vars".DO6.iCounterIn, iCounterOut := "PLC8_910A4_8DI_8DO_DO_Vars".DO6.iCounterOut, xOutput => "PLC8_910A4_8DI_8DO_DO_Vars".DO6.xOutput)
   END_RUNG
   RUNG wire#powerrail
      Contact( "PLC8_910A4_8DI_8DO_DO_Vars".DO6.xOutput )
      Coil( "DO8.04.06" )
   END_RUNG
   // the same network as SCL:
   "DOvar"(iFuncSystem := "PLC8_910A4_8DI_8DO_DO_Vars".DO6.iFuncSystemID,
           iFuncVar := "PLC8_910A4_8DI_8DO_DO_Vars".DO6.iFuncVar,
           xOutput => "PLC8_910A4_8DI_8DO_DO_Vars".DO6.xInput);
   "DOadv"(xInput := "PLC8_910A4_8DI_8DO_DO_Vars".DO6.xInput,
           xInversion := "PLC8_910A4_8DI_8DO_DO_Vars".DO6.xInversion,
           cMOA := "PLC8_910A4_8DI_8DO_DO_Vars".DO6.cMOA,
           xMemoryOut := "PLC8_910A4_8DI_8DO_DO_Vars".DO6.xMemoryOut,
           xMemoryIn := "PLC8_910A4_8DI_8DO_DO_Vars".DO6.xMemoryIn,
           cMemory := "PLC8_910A4_8DI_8DO_DO_Vars".DO6.cMemory,
           iCounterIn := "PLC8_910A4_8DI_8DO_DO_Vars".DO6.iCounterIn,
           iCounterOut := "PLC8_910A4_8DI_8DO_DO_Vars".DO6.iCounterOut,
           xOutput => "PLC8_910A4_8DI_8DO_DO_Vars".DO6.xOutput);
   "DO8.04.06" := "PLC8_910A4_8DI_8DO_DO_Vars".DO6.xOutput;
END_REGION

REGION Network 15: DQa6
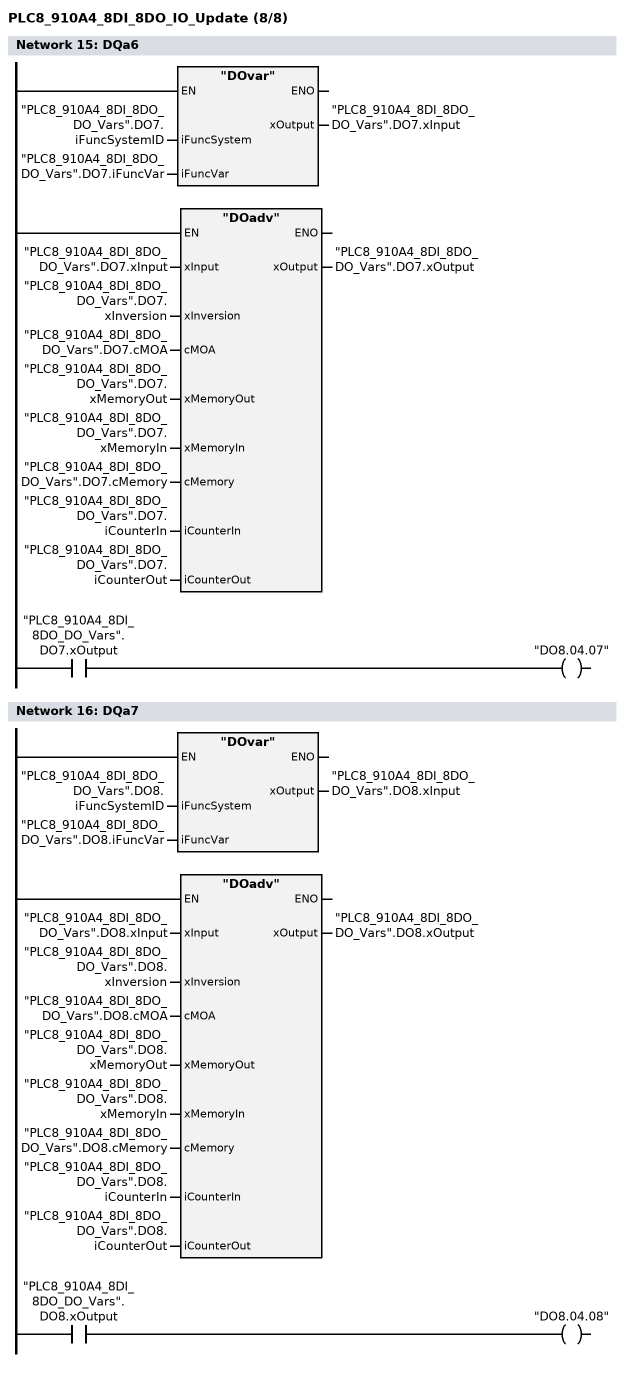
   RUNG wire#powerrail
      "DOvar"(iFuncSystem := "PLC8_910A4_8DI_8DO_DO_Vars".DO7.iFuncSystemID, iFuncVar := "PLC8_910A4_8DI_8DO_DO_Vars".DO7.iFuncVar, xOutput => "PLC8_910A4_8DI_8DO_DO_Vars".DO7.xInput)
   END_RUNG
   RUNG wire#powerrail
      "DOadv"(xInput := "PLC8_910A4_8DI_8DO_DO_Vars".DO7.xInput, xInversion := "PLC8_910A4_8DI_8DO_DO_Vars".DO7.xInversion, cMOA := "PLC8_910A4_8DI_8DO_DO_Vars".DO7.cMOA, xMemoryOut := "PLC8_910A4_8DI_8DO_DO_Vars".DO7.xMemoryOut, xMemoryIn := "PLC8_910A4_8DI_8DO_DO_Vars".DO7.xMemoryIn, cMemory := "PLC8_910A4_8DI_8DO_DO_Vars".DO7.cMemory, iCounterIn := "PLC8_910A4_8DI_8DO_DO_Vars".DO7.iCounterIn, iCounterOut := "PLC8_910A4_8DI_8DO_DO_Vars".DO7.iCounterOut, xOutput => "PLC8_910A4_8DI_8DO_DO_Vars".DO7.xOutput)
   END_RUNG
   RUNG wire#powerrail
      Contact( "PLC8_910A4_8DI_8DO_DO_Vars".DO7.xOutput )
      Coil( "DO8.04.07" )
   END_RUNG
   // the same network as SCL:
   "DOvar"(iFuncSystem := "PLC8_910A4_8DI_8DO_DO_Vars".DO7.iFuncSystemID,
           iFuncVar := "PLC8_910A4_8DI_8DO_DO_Vars".DO7.iFuncVar,
           xOutput => "PLC8_910A4_8DI_8DO_DO_Vars".DO7.xInput);
   "DOadv"(xInput := "PLC8_910A4_8DI_8DO_DO_Vars".DO7.xInput,
           xInversion := "PLC8_910A4_8DI_8DO_DO_Vars".DO7.xInversion,
           cMOA := "PLC8_910A4_8DI_8DO_DO_Vars".DO7.cMOA,
           xMemoryOut := "PLC8_910A4_8DI_8DO_DO_Vars".DO7.xMemoryOut,
           xMemoryIn := "PLC8_910A4_8DI_8DO_DO_Vars".DO7.xMemoryIn,
           cMemory := "PLC8_910A4_8DI_8DO_DO_Vars".DO7.cMemory,
           iCounterIn := "PLC8_910A4_8DI_8DO_DO_Vars".DO7.iCounterIn,
           iCounterOut := "PLC8_910A4_8DI_8DO_DO_Vars".DO7.iCounterOut,
           xOutput => "PLC8_910A4_8DI_8DO_DO_Vars".DO7.xOutput);
   "DO8.04.07" := "PLC8_910A4_8DI_8DO_DO_Vars".DO7.xOutput;
END_REGION

REGION Network 16: DQa7
   RUNG wire#powerrail
      "DOvar"(iFuncSystem := "PLC8_910A4_8DI_8DO_DO_Vars".DO8.iFuncSystemID, iFuncVar := "PLC8_910A4_8DI_8DO_DO_Vars".DO8.iFuncVar, xOutput => "PLC8_910A4_8DI_8DO_DO_Vars".DO8.xInput)
   END_RUNG
   RUNG wire#powerrail
      "DOadv"(xInput := "PLC8_910A4_8DI_8DO_DO_Vars".DO8.xInput, xInversion := "PLC8_910A4_8DI_8DO_DO_Vars".DO8.xInversion, cMOA := "PLC8_910A4_8DI_8DO_DO_Vars".DO8.cMOA, xMemoryOut := "PLC8_910A4_8DI_8DO_DO_Vars".DO8.xMemoryOut, xMemoryIn := "PLC8_910A4_8DI_8DO_DO_Vars".DO8.xMemoryIn, cMemory := "PLC8_910A4_8DI_8DO_DO_Vars".DO8.cMemory, iCounterIn := "PLC8_910A4_8DI_8DO_DO_Vars".DO8.iCounterIn, iCounterOut := "PLC8_910A4_8DI_8DO_DO_Vars".DO8.iCounterOut, xOutput => "PLC8_910A4_8DI_8DO_DO_Vars".DO8.xOutput)
   END_RUNG
   RUNG wire#powerrail
      Contact( "PLC8_910A4_8DI_8DO_DO_Vars".DO8.xOutput )
      Coil( "DO8.04.08" )
   END_RUNG
   // the same network as SCL:
   "DOvar"(iFuncSystem := "PLC8_910A4_8DI_8DO_DO_Vars".DO8.iFuncSystemID,
           iFuncVar := "PLC8_910A4_8DI_8DO_DO_Vars".DO8.iFuncVar,
           xOutput => "PLC8_910A4_8DI_8DO_DO_Vars".DO8.xInput);
   "DOadv"(xInput := "PLC8_910A4_8DI_8DO_DO_Vars".DO8.xInput,
           xInversion := "PLC8_910A4_8DI_8DO_DO_Vars".DO8.xInversion,
           cMOA := "PLC8_910A4_8DI_8DO_DO_Vars".DO8.cMOA,
           xMemoryOut := "PLC8_910A4_8DI_8DO_DO_Vars".DO8.xMemoryOut,
           xMemoryIn := "PLC8_910A4_8DI_8DO_DO_Vars".DO8.xMemoryIn,
           cMemory := "PLC8_910A4_8DI_8DO_DO_Vars".DO8.cMemory,
           iCounterIn := "PLC8_910A4_8DI_8DO_DO_Vars".DO8.iCounterIn,
           iCounterOut := "PLC8_910A4_8DI_8DO_DO_Vars".DO8.iCounterOut,
           xOutput => "PLC8_910A4_8DI_8DO_DO_Vars".DO8.xOutput);
   "DO8.04.08" := "PLC8_910A4_8DI_8DO_DO_Vars".DO8.xOutput;
END_REGION
END_FUNCTION
